// SIMATIC S7-200 SMART project (STEP 7-Micro/WIN SMART), CPU SR40

SYMBOL_TABLE 系统符号
Always_On        SM0.0    // 始终接通
First_Scan_On    SM0.1    // 仅在第一个扫描周期时接通
Clock_1s         SM0.5    // 针对 1 s 的周期时间，时钟脉冲接通 0.5 s，断开 0.5 s.
END_SYMBOL_TABLE

ORGANIZATION_BLOCK MAIN:OB1
TITLE=程序注释
BEGIN
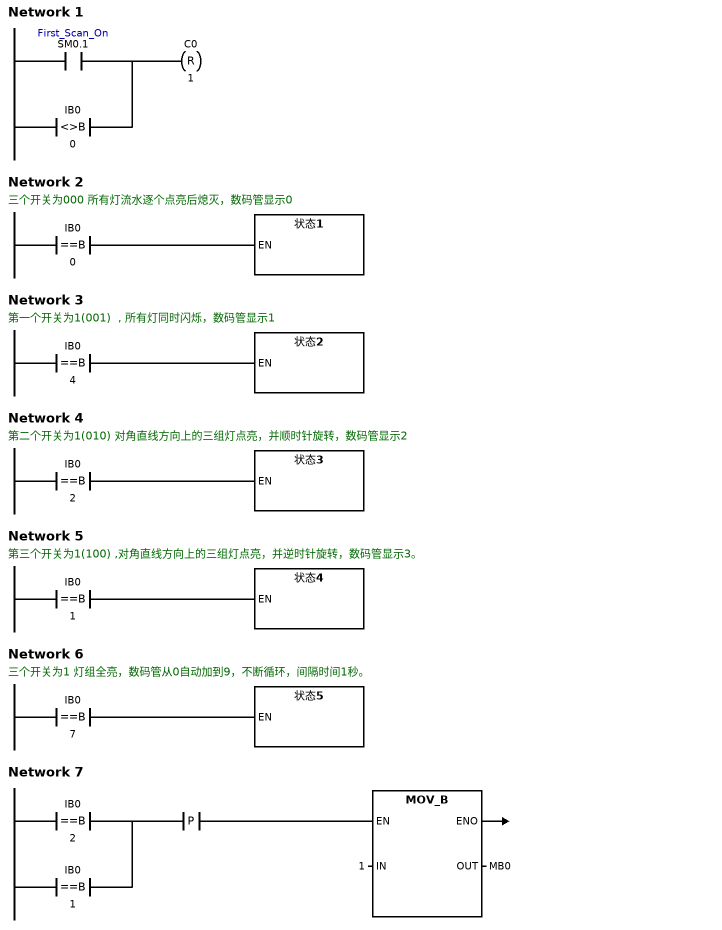
Network 1
LD     First_Scan_On:SM0.1
OB<>   IB0, 0
R      C0, 1
Network 2
// 三个开关为000 所有灯流水逐个点亮后熄灭，数码管显示0
LDB=   IB0, 0
CALL   状态1:SBR0
Network 3
// 第一个开关为1(001)  , 所有灯同时闪烁，数码管显示1
LDB=   IB0, 4
CALL   状态2:SBR1
Network 4
// 第二个开关为1(010) 对角直线方向上的三组灯点亮，并顺时针旋转，数码管显示2
LDB=   IB0, 2
CALL   状态3:SBR2
Network 5
//  第三个开关为1(100) ,对角直线方向上的三组灯点亮，并逆时针旋转，数码管显示3。
LDB=   IB0, 1
CALL   状态4:SBR3
Network 6
// 三个开关为1 灯组全亮，数码管从0自动加到9，不断循环，间隔时间1秒。
LDB=   IB0, 7
CALL   状态5:SBR4
Network 7
LDB=   IB0, 2
OB=    IB0, 1
EU
MOVB   1, MB0
END_ORGANIZATION_BLOCK

SUBROUTINE_BLOCK 状态1:SBR0
TITLE=所有灯流水逐个点亮后熄灭，数码管显示0
BEGIN
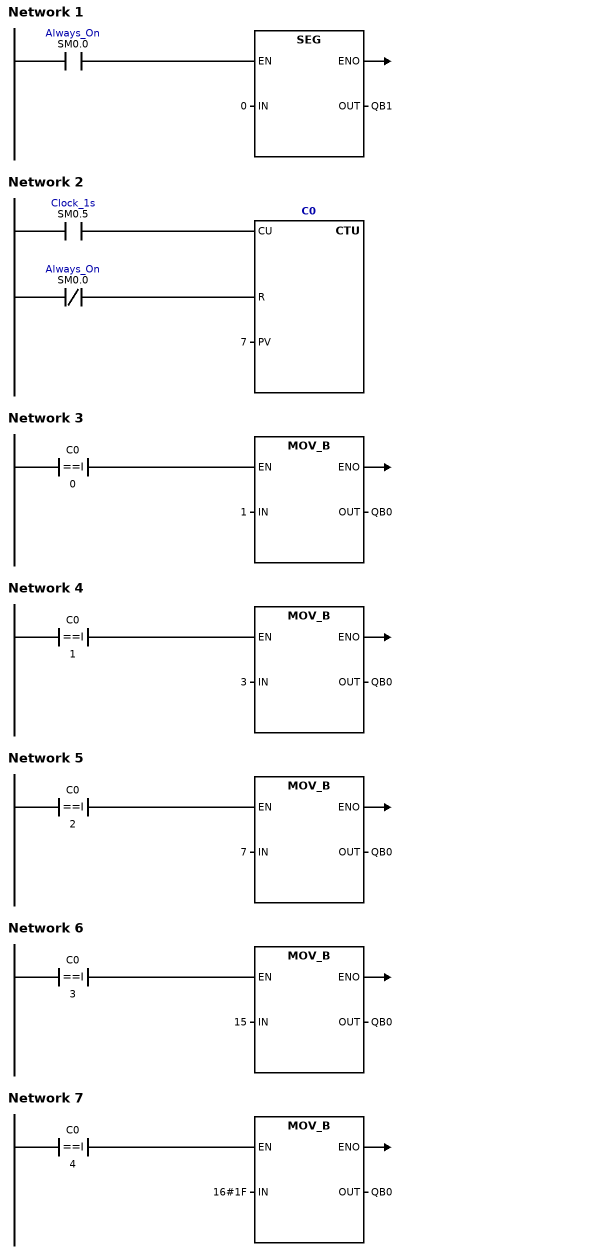
Network 1
LD     Always_On:SM0.0
SEG    0, QB1
Network 2
LD     Clock_1s:SM0.5
LDN    Always_On:SM0.0
CTU    C0, 7
Network 3
LDW=   C0, 0
MOVB   1, QB0
Network 4
LDW=   C0, 1
MOVB   3, QB0
Network 5
LDW=   C0, 2
MOVB   7, QB0
Network 6
LDW=   C0, 3
MOVB   15, QB0
Network 7
LDW=   C0, 4
MOVB   16#1F, QB0
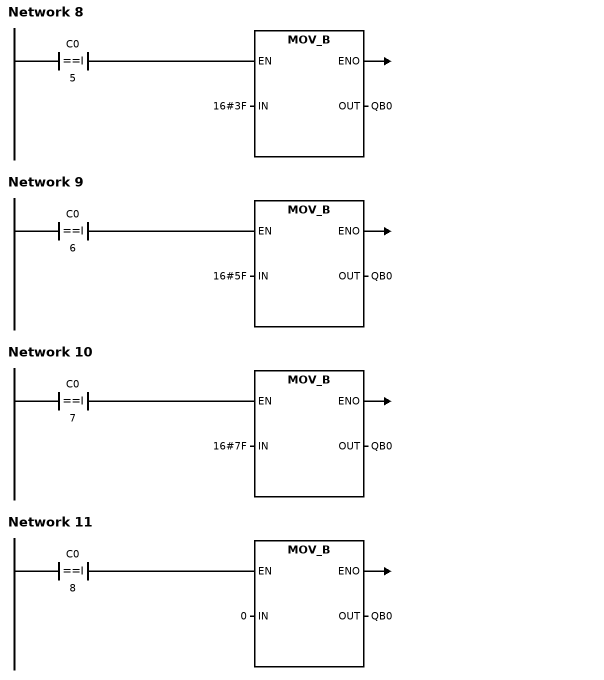
Network 8
LDW=   C0, 5
MOVB   16#3F, QB0
Network 9
LDW=   C0, 6
MOVB   16#5F, QB0
Network 10
LDW=   C0, 7
MOVB   16#7F, QB0
Network 11
LDW=   C0, 8
MOVB   0, QB0
END_SUBROUTINE_BLOCK

SUBROUTINE_BLOCK 状态2:SBR1
TITLE=子程序注释
BEGIN
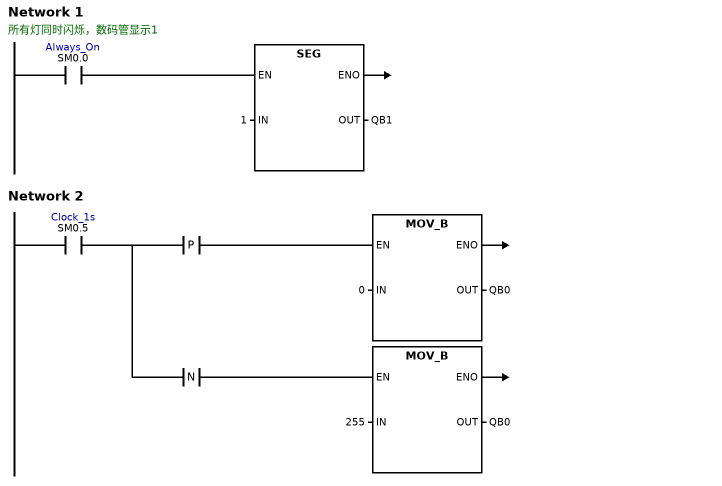
Network 1
// 所有灯同时闪烁，数码管显示1
LD     Always_On:SM0.0
SEG    1, QB1
Network 2
LD     Clock_1s:SM0.5
LPS
EU
MOVB   0, QB0
LPP
ED
MOVB   255, QB0
END_SUBROUTINE_BLOCK

SUBROUTINE_BLOCK 状态3:SBR2
TITLE=子程序注释
BEGIN
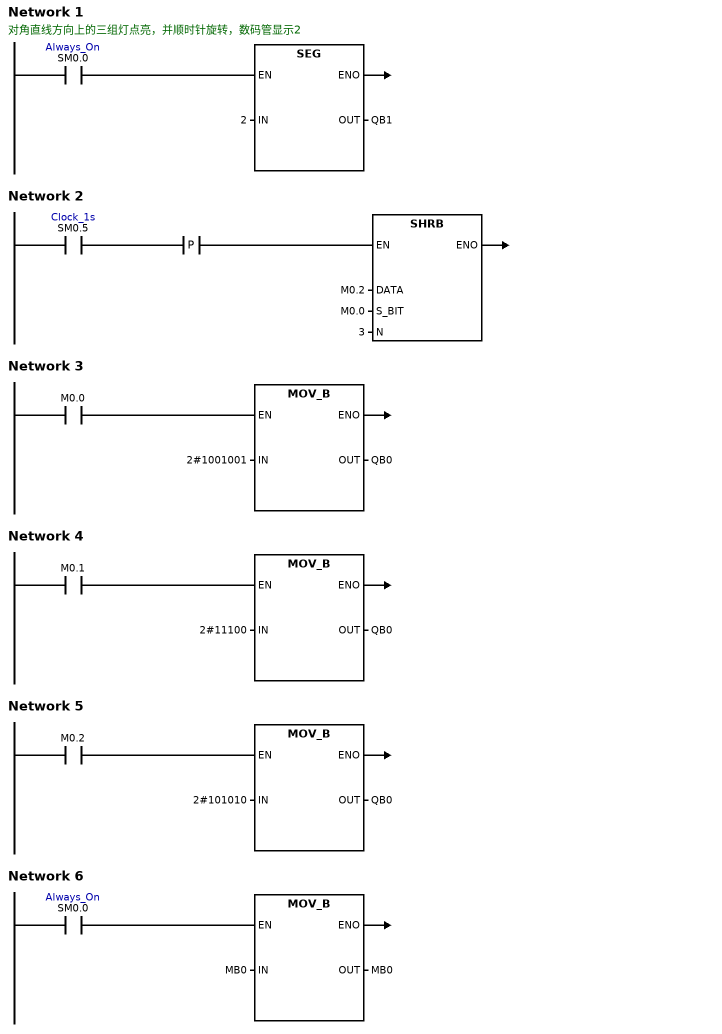
Network 1
// 对角直线方向上的三组灯点亮，并顺时针旋转，数码管显示2
LD     Always_On:SM0.0
SEG    2, QB1
Network 2
LD     Clock_1s:SM0.5
EU
SHRB   M0.2, M0.0, 3
Network 3
LD     M0.0
MOVB   2#1001001, QB0
Network 4
LD     M0.1
MOVB   2#11100, QB0
Network 5
LD     M0.2
MOVB   2#101010, QB0
Network 6
LD     Always_On:SM0.0
MOVB   MB0, MB0
END_SUBROUTINE_BLOCK

SUBROUTINE_BLOCK 状态4:SBR3
TITLE=对角直线方向上的三组灯点亮，并逆时针旋转，数码管显示3。
BEGIN
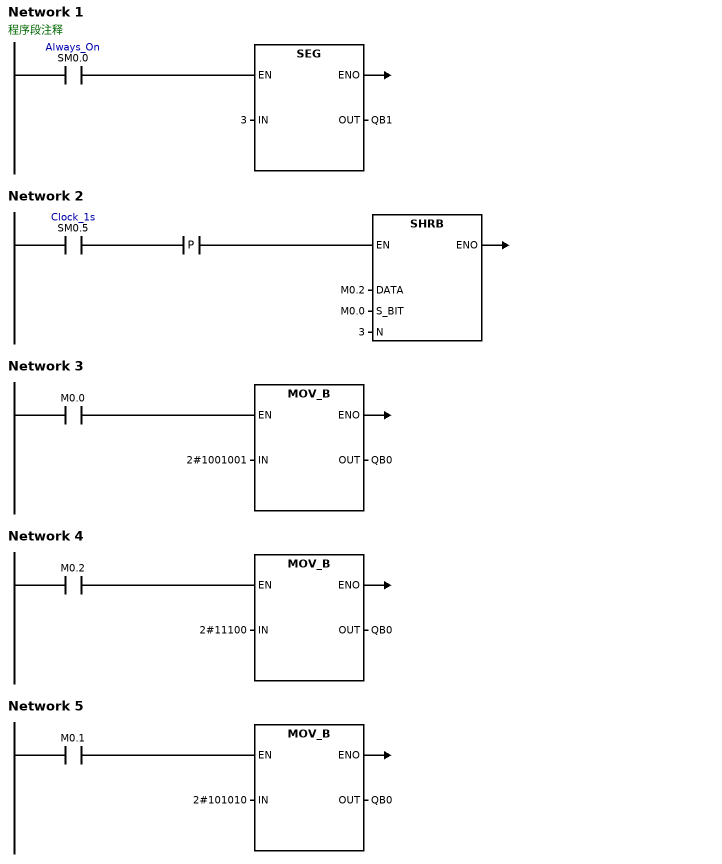
Network 1
// 程序段注释
LD     Always_On:SM0.0
SEG    3, QB1
Network 2
LD     Clock_1s:SM0.5
EU
SHRB   M0.2, M0.0, 3
Network 3
LD     M0.0
MOVB   2#1001001, QB0
Network 4
LD     M0.2
MOVB   2#11100, QB0
Network 5
LD     M0.1
MOVB   2#101010, QB0
END_SUBROUTINE_BLOCK

SUBROUTINE_BLOCK 状态5:SBR4
TITLE=灯组全亮，数码管从0自动加到9，不断循环，间隔时间1秒。
BEGIN
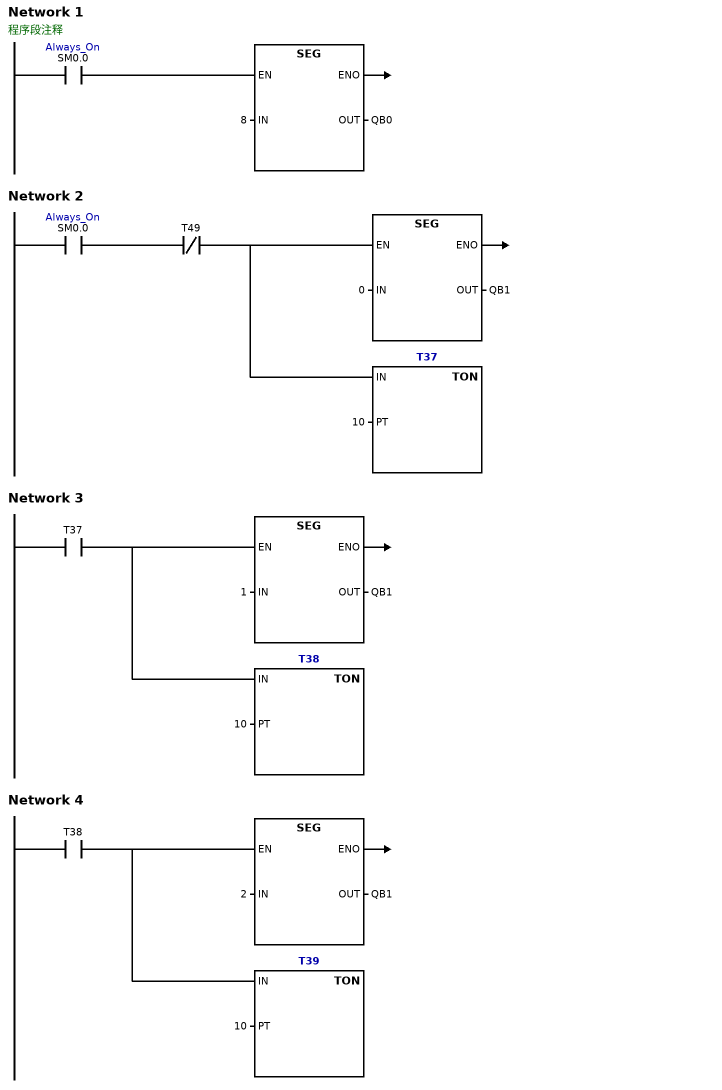
Network 1
// 程序段注释
LD     Always_On:SM0.0
SEG    8, QB0
Network 2
LD     Always_On:SM0.0
AN     T49
SEG    0, QB1
TON    T37, 10
Network 3
LD     T37
SEG    1, QB1
TON    T38, 10
Network 4
LD     T38
SEG    2, QB1
TON    T39, 10
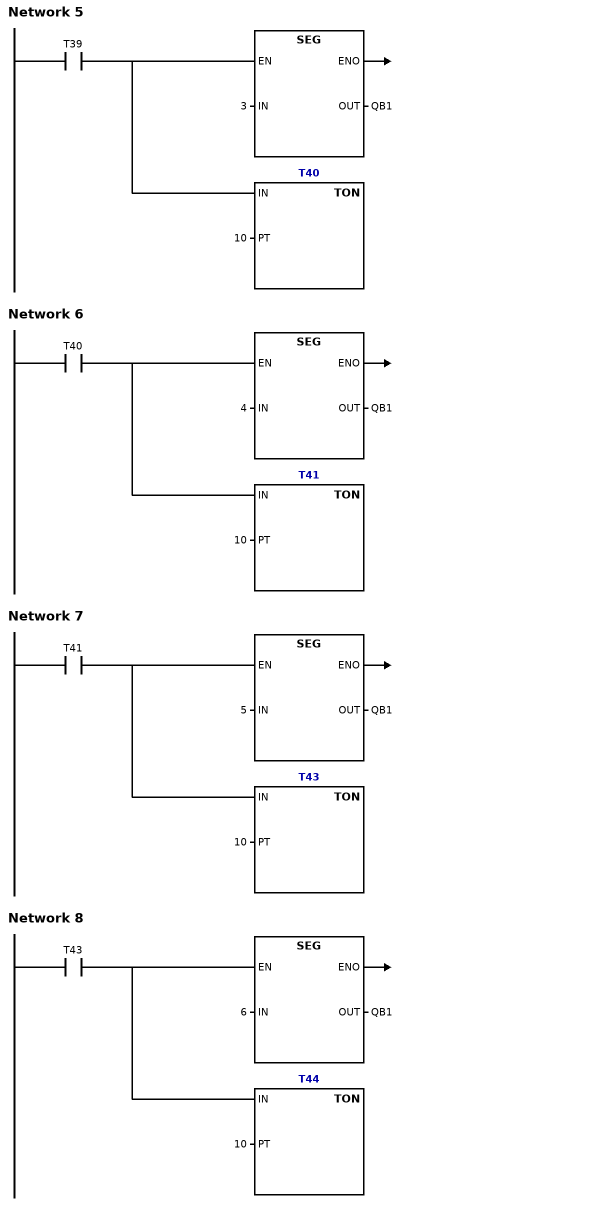
Network 5
LD     T39
SEG    3, QB1
TON    T40, 10
Network 6
LD     T40
SEG    4, QB1
TON    T41, 10
Network 7
LD     T41
SEG    5, QB1
TON    T43, 10
Network 8
LD     T43
SEG    6, QB1
TON    T44, 10
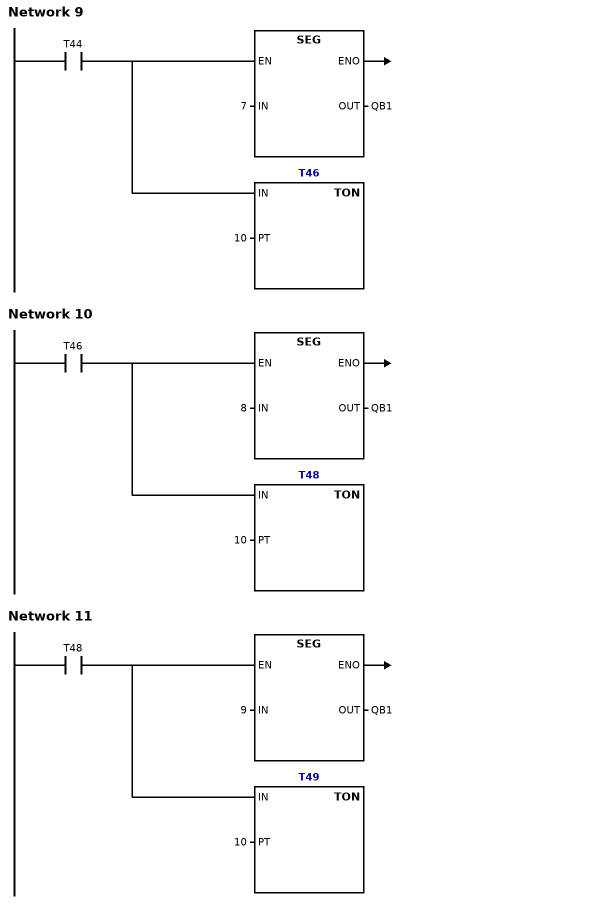
Network 9
LD     T44
SEG    7, QB1
TON    T46, 10
Network 10
LD     T46
SEG    8, QB1
TON    T48, 10
Network 11
LD     T48
SEG    9, QB1
TON    T49, 10
Network 12
// 程序段注释
END_SUBROUTINE_BLOCK
